// get postion of myself
rPosOnTrack := iMover.getAxisRef.NcToPlc.ModuloActPos;

// go through the list and search the mover in front
THIS^.fbMovers.ResetIterator();
WHILE THIS^.fbMovers.HasNextObject() DO
	IF ToMover(THIS^.fbMovers.GetNextObject(), iTempMover) THEN
		// if Mover is myself, skipp
		IF iTempMover <> iMover THEN
			// calc distance to Mover in positive direction
			rTempDistBetween := FUN_GetDistToPosModulo(ActualPosition := rPosOnTrack, TargedPosition := iTempMover.getAxisRef.NcToPlc.ModuloActPos, Modulo := TrackLength);
	
	
			// check if Mover is closer then last one
			IF rFoundDistBetween > rTempDistBetween THEN 
				rFoundDistBetween := rTempDistBetween;
				iFoundMover := iTempMover;
			END_IF
		END_IF
	END_IF
END_WHILE

getMoverInFront := iFoundMover;
END_METHOD

METHOD getStationInFront : I_XTS_Station
VAR_INPUT
	iStation	: I_XTS_Station;
END_VAR
VAR
	rPosOnTrack: LREAL;
	
	iTempStation : I_XTS_Station;
	rTempPosOnTrack: LREAL;
	rTempDistBetween : LREAL;
	
	rFoundDistBetween : LREAL := TrackLength;
	iFoundStation	: I_XTS_Station;
END_VAR
// get postion of myself
rPosOnTrack := iStation.PositionOnTrack;

// go through the list and search the station in front
THIS^.fbStations.ResetIterator();
WHILE THIS^.fbStations.HasNextObject() DO
	IF ToStation(THIS^.fbStations.GetNextObject(), iTempStation) THEN
		// calc distance to Station
		rTempDistBetween := iTempStation.PositionOnTrack - rPosOnTrack;		
		
		// if Station is behinde me or it is myself -> add Modulo
		IF rTempDistBetween <= 0 THEN 
			rTempDistBetween := rTempDistBetween + TrackLength;			
		END_IF

		// check if Station is closer then last one
		IF rFoundDistBetween > rTempDistBetween THEN 
			rFoundDistBetween := rTempDistBetween;
			iFoundStation := iTempStation;
		END_IF
		
	END_IF
END_WHILE

getStationInFront := iFoundStation;
END_METHOD

METHOD Initialize : HRESULT
VAR
	hr : HRESULT;
END_VAR
IF THIS^.iEnvironment.Initialize() = S_OK THEN
	hr := GetMostSignificant(hr, fbMovers.Initialize());	
	hr := GetMostSignificant(hr, iGroup.Initialize());	
	hr := GetMostSignificant(hr, fbStations.Initialize());	
	hr := GetMostSignificant(hr, fbZone.Initialize());	
	hr := GetMostSignificant(hr, fbTrigger.Initialize());	
ELSE
	hr := S_PENDING;
END_IF	


THIS^.bInitDone := (hr = S_OK);
Initialize:= hr;
END_METHOD

{attribute 'monitoring':='call'}
PROPERTY Initialized : BOOL
GET
Initialized := bInitDone;
END_GET
END_PROPERTY

METHOD LinkEnvironment : HRESULT
VAR_INPUT
	iEnvironment	: CHALET_BaseComponents.I_CH_Object;
END_VAR

VAR
	iXtsEnvironment : I_Xts_Environment;
END_VAR
IF iEnvironment <> 0 AND_THEN __QUERYINTERFACE(iEnvironment, iXtsEnvironment) THEN
	THIS^.iEnvironment := iXtsEnvironment;
END_IF
END_METHOD

METHOD LinkGroup : HRESULT
VAR_INPUT
	Group	: CHALET_BaseComponents.I_CH_Object;
END_VAR

VAR
	iXtsGroup : I_XTS_Group;
END_VAR
IF Group <> 0 AND_THEN __QUERYINTERFACE(Group, iXtsGroup) THEN
	THIS^.iGroup := iXtsGroup;
END_IF
END_METHOD

{attribute 'monitoring':='call'}
PROPERTY Movers : CHALET_BaseComponents.I_CH_LIST
GET
Movers := THIS^.fbMovers;
END_GET
END_PROPERTY

METHOD RegisterMover : HRESULT
VAR_INPUT
	Mover	: CHALET_BaseComponents.I_CH_Object;
END_VAR

VAR
	iXtsMover : I_XTS_Mover;
END_VAR
IF Mover <> 0 AND_THEN __QUERYINTERFACE(Mover,iXtsMover) THEN
	THIS^.fbMovers.AddObject(Mover);
END_IF
END_METHOD

METHOD RegisterStation : HRESULT
VAR_INPUT
	Station	: CHALET_BaseComponents.I_CH_Object;
END_VAR

VAR
	iStation : I_XTS_Station;
END_VAR
IF Station <> 0 AND_THEN __QUERYINTERFACE(Station,iStation) THEN
	THIS^.fbStations.AddObject(Station);
END_IF
END_METHOD

METHOD RegisterTrigger : HRESULT
VAR_INPUT
	Trigger	: CHALET_BaseComponents.I_CH_Object;
END_VAR
VAR
	iTrigger : I_XTS_Trigger;
END_VAR
IF Trigger <> 0 AND_THEN __QUERYINTERFACE(Trigger,iTrigger) THEN
	THIS^.fbTrigger.AddObject(Trigger);
END_IF
END_METHOD

METHOD RegisterZone : HRESULT
VAR_INPUT
	Zone	: CHALET_BaseComponents.I_CH_Object;
END_VAR
VAR
	iZone : I_XTS_Zone;
END_VAR
IF Zone <> 0 AND_THEN __QUERYINTERFACE(Zone,iZone) THEN
	THIS^.fbZone.AddObject(Zone);
END_IF
END_METHOD

{warning 'add method implementation '}
METHOD Reset : HRESULT
END_METHOD

METHOD Station : I_XTS_Station_PLC
VAR_INPUT
	sLUID	: STRING;
END_VAR
//IF no station was found, INTERFACE is 0 -> can generate fatal error
__QUERYINTERFACE(THIS^.fbStations.FindLUID(sLUID),Station);
END_METHOD

PROPERTY Stations : CHALET_BaseComponents.I_CH_LIST
GET
Stations := THIS^.fbStations;
END_GET
END_PROPERTY

{attribute 'monitoring':='call'}
PROPERTY SuppressAllDynamicsChanges : BOOL
SET
VAR
	iTempStationPlc : I_XTS_Station_PLC;
END_VAR
// go through the list and write request to it
THIS^.fbStations.ResetIterator();
WHILE THIS^.fbStations.HasNextObject() DO
	IF ToStation_PLC(THIS^.fbStations.GetNextObject(), iTempStationPlc) THEN
		iTempStationPlc.SuppressDynamicsChange := SuppressAllDynamicsChanges;
	END_IF
END_WHILE
END_SET
END_PROPERTY

{attribute 'monitoring':='call'}
PROPERTY TrackLength : LREAL
GET
TrackLength := THIS^.iEnvironment.TrackLength;
END_GET
END_PROPERTY

METHOD Update : HRESULT
VAR_INPUT
END_VAR
VAR
	hr : HRESULT;
END_VAR
hr := S_OK;

hr := GetMostSignificant(hr, THIS^.Enabling());	
hr := GetMostSignificant(hr, THIS^.Disabling());	

THIS^.fbFeedback.HR := hr;

hr := GetMostSignificant(hr, THIS^.fbMovers.Update());	
hr := GetMostSignificant(hr, THIS^.fbStations.Update());	
hr := GetMostSignificant(hr, THIS^.fbZone.Update());	
hr := GetMostSignificant(hr, THIS^.fbTrigger.Update());	

//zzz Todo vllt könnte hier später das CH_Object verwendet werden
hr := GetMostSignificant(hr, THIS^.iGroup.Update());	
hr := GetMostSignificant(hr, THIS^.iEnvironment.Update());	

Update:= hr;
END_METHOD

END_FUNCTION_BLOCK

// COMPENENTs/System/I_XTS_System_PLC
INTERFACE I_XTS_System_PLC

METHOD Disable : I_CH_Feedback
VAR_INPUT
END_VAR
END_METHOD

{attribute 'monitoring':='call'}
PROPERTY Disabled : Bool
GET
END_GET
END_PROPERTY

METHOD Enable : I_CH_Feedback
VAR_INPUT
END_VAR
END_METHOD

{attribute 'monitoring':='call'}
PROPERTY Enabled : Bool
GET
END_GET
END_PROPERTY

{attribute 'monitoring':='call'}
PROPERTY Feedback : CHALET_BaseComponents.I_CH_Feedback
GET
END_GET
END_PROPERTY

METHOD Initialize : HRESULT
VAR_INPUT
END_VAR
END_METHOD

{attribute 'monitoring':='call'}
PROPERTY Initialized : BOOL
GET
END_GET
END_PROPERTY

METHOD Reset : HRESULT
VAR_INPUT
END_VAR
END_METHOD

METHOD Station : I_XTS_Station_PLC
VAR_INPUT
	sLUID : STRING;
END_VAR
END_METHOD

PROPERTY SuppressAllDynamicsChanges : BOOL
SET
END_SET
END_PROPERTY

{attribute 'monitoring':='call'}
PROPERTY TrackLength : LREAL
GET
END_GET
END_PROPERTY

METHOD Update : HRESULT
VAR_INPUT
END_VAR
END_METHOD

END_INTERFACE
